// TwinCAT 3 PLC project SortingMashine
// ProgramVersion: 3.1.4023.0
// libraries:
//   Tc2_Standard, * (Beckhoff Automation GmbH)
//   Tc2_System, * (Beckhoff Automation GmbH)
//   Tc3_Module, * (Beckhoff Automation GmbH)
// project tree:
//   DUTs/ Material_Type.TcDUT, Positions.TcDUT
//   / GlobalTextList.TcGTLO, PlcTask.TcTTO, Visualization Manager.TcVMO (not stored)
//   POUs/ FB_Axes.TcPOU, FB_Box.TcPOU, FB_Gate.TcPOU, MAIN.TcPOU, Mashine.TcPOU
//   VISUs/ Visualization.TcVIS
// real-time tasks:
//   TASK PlcTask: cycle T#10ms, priority 20, ADS port 350

CONFIGURATION SortingMashine
    RESOURCE PLC ON TwinCAT3
        TASK PlcTask(INTERVAL := T#10ms, PRIORITY := 20);
        PROGRAM MAIN WITH PlcTask : MAIN;
    END_RESOURCE
END_CONFIGURATION

// ---- DUTs/Material_Type.TcDUT
{attribute 'qualified_only'}
{attribute 'strict'}
TYPE Material_Type :
(
	Plastic := 0,
	Metal :=1
);
END_TYPE

// ---- DUTs/Positions.TcDUT
{attribute 'qualified_only'}
{attribute 'strict'}
TYPE Positions :
(
	First := 180,
	Second:=148,
	Third:=116,
	Forth:=84
);
END_TYPE

// ---- POUs/MAIN.TcPOU
PROGRAM MAIN
VAR
	Mashine1Boxes:ARRAY[1..4] OF FB_Box;
	Mashine2Boxes:ARRAY[1..4] OF FB_Box;
	MyMashine1:Mashine;
	MyMashine2:Mashine;
END_VAR

Mashine1Boxes[1](material:=Material_Type.Plastic);
Mashine1Boxes[2](material:=Material_Type.Metal);
Mashine1Boxes[3](material:=Material_Type.Plastic);
Mashine1Boxes[4](material:=Material_Type.Metal);
Mashine2Boxes[1](material:=Material_Type.Metal);
Mashine2Boxes[2](material:=Material_Type.Plastic);
Mashine2Boxes[3](material:=Material_Type.Metal);
Mashine2Boxes[4](material:=Material_Type.Plastic);

MyMashine1(Box:=Mashine1Boxes);
MyMashine2(Box:=Mashine2Boxes);

END_PROGRAM

// ---- POUs/FB_Box.TcPOU
FUNCTION_BLOCK FB_Box
VAR_INPUT
		material : Material_Type;
		PositionHOZ : INT;
		PositionVTK : INT;
END_VAR
VAR_OUTPUT
END_VAR
VAR
	IsMetal:BOOL;
END_VAR

M_Identify_Material();

METHOD M_Identify_Material : BOOL
VAR_INPUT
END_VAR
IF material=Material_Type.Metal THEN
	IsMetal:=TRUE;
ELSE
	IsMetal:=FALSE;
END_IF
END_METHOD

END_FUNCTION_BLOCK

// ---- POUs/Mashine.TcPOU
FUNCTION_BLOCK Mashine 
VAR_INPUT
	Box:REFERENCE TO ARRAY[1..4] OF FB_Box;
END_VAR
VAR_OUTPUT
END_VAR
VAR
	Current:INT:=1;
	MyGate:FB_Gate;
	FirstAxes:FB_Axes;
	SecondAxes:FB_Axes;
	Step_Stat:INT;
	Step_Stat2:INT;
	Step_Stat3:INT;
END_VAR

CASE Step_Stat OF
	
	0:
		IF OpenGate() THEN
			Step_Stat:=Step_Stat+1;
		END_IF
	1:
		IF MoveOut(Box[Current]) THEN
			Step_Stat:=Step_Stat+1;
		END_IF
	2:
		IF CloseGate()  THEN
			Step_Stat:=Step_Stat+1;
		END_IF
	3:
		IF MoveToFirstPosition(Box[Current])  THEN
			Step_Stat:=Step_Stat+1;
		END_IF
	4:
		IF NOT Box[Current].IsMetal THEN
			IF ExtendFirstAxes(Box[Current]) THEN
				IF Current <4 THEN
					Current:=Current+1;
					Step_Stat:=0;
				ELSE
					Step_Stat:=7;
				END_IF
			END_IF
		ELSE
			Step_Stat:=Step_Stat+1;
		END_IF
	5:
		IF MoveToSecondPosition(Box[Current]) THEN
			Step_Stat:=Step_Stat+1;
		END_IF
	6:
		IF Box[Current].IsMetal THEN
			IF ExtendSecondAxes(Box[Current]) THEN
				IF Current <4 THEN
					Current:=Current+1;
					Step_Stat:=0;
				ELSE
					Step_Stat:=7;
				END_IF
			END_IF
		END_IF
	7://End
		
END_CASE

METHOD CloseGate : BOOL
VAR_INPUT
END_VAR
IF MyGate.GateStat = TRUE THEN
MyGate.GateTimer(IN:=TRUE,PT:=T#1S);	
	IF MyGate.GatePosition > 0 THEN
		MyGate.GatePosition:=MyGate.GatePosition-1;
	END_IF
	IF MyGate.GateTimer.Q THEN		
		MyGate.GateTimer(IN:=FALSE);	
		MyGate.GateStat:=FALSE;
		CloseGate:=TRUE;	
	END_IF	
END_IF
END_METHOD

METHOD ExtendFirstAxes : BOOL
VAR_INPUT
	Box:reference to FB_Box;
END_VAR
CASE FirstAxes.Axes_Step OF
	0:
		IF  FirstAxes.AxesPosition > -55 THEN
			FirstAxes.AxesPosition:= FirstAxes.AxesPosition-1;
			Box.PositionVTK:=Box.PositionVTK-4;
			IF  FirstAxes.AxesPosition <= -55 AND Box.PositionVTK <= -200 THEN
				FirstAxes.Axes_Step:=FirstAxes.Axes_Step+1;
			END_IF
		END_IF		
	1: 
		IF  FirstAxes.AxesPosition < 0 THEN	
			FirstAxes.AxesPosition:= FirstAxes.AxesPosition+1;
			IF  FirstAxes.AxesPosition = 0 THEN
				ExtendFirstAxes:=TRUE;
				FirstAxes.Axes_Step:=0;
			END_IF		
		END_IF
END_CASE	







//IF FirstAxes.Extended = FALSE THEN
//	IF  FirstAxes.AxesPosition > -55 THEN
//		 FirstAxes.AxesPosition:= FirstAxes.AxesPosition-1;
//	END_IF	
	
//	IF  FirstAxes.AxesPosition = -55 THEN
		
//			FirstAxes.Extended:=TRUE;
//		 	FirstAxes.AxesTimer(IN:=TRUE,PT:=T#500MS);
//		IF FirstAxes.AxesTimer.Q AND  FirstAxes.Extended:=TRUE THEN
			
//			IF  FirstAxes.AxesPosition < 0 THEN
//				 FirstAxes.AxesPosition:= FirstAxes.AxesPosition+1;
//			END_IF
	
//			IF  FirstAxes.AxesPosition = 0 THEN
//				FirstAxes.AxesTimer(IN:=FALSE);
//				FirstAxes.Extended:=FALSE;
//			END_IF
			
//		END_IF
		
//	END_IF
	
//END_IF
END_METHOD

METHOD ExtendSecondAxes : BOOL
VAR_INPUT
	Box:REFERENCE TO FB_Box;
END_VAR
CASE SecondAxes.Axes_Step OF
	0: 
		IF  SecondAxes.AxesPosition > -55 THEN
			SecondAxes.AxesPosition:= SecondAxes.AxesPosition-1;
			Box.PositionVTK:=Box.PositionVTK-4;
			IF  SecondAxes.AxesPosition <= -55 AND Box.PositionVTK <= -200 THEN
				SecondAxes.Axes_Step:=SecondAxes.Axes_Step+1;
			END_IF
		END_IF		
	1: 
		IF  SecondAxes.AxesPosition < 0 THEN	
			SecondAxes.AxesPosition:= SecondAxes.AxesPosition+1;
			IF  SecondAxes.AxesPosition = 0 THEN
				ExtendSecondAxes:=TRUE;
				SecondAxes.Axes_Step:=0;
			END_IF		
		END_IF
END_CASE
END_METHOD

METHOD MoveOut : BOOL
VAR_INPUT
	Box: reference to FB_Box;
END_VAR
IF Box.PositionHOZ < 50 THEN
Box.PositionHOZ:=Box.PositionHOZ+1;	
	IF Box.PositionHOZ = 50 THEN
		MoveOut:=TRUE;		
	END_IF
ELSIF Box.PositionHOZ = 50 THEN
	MoveOut:=TRUE;
END_IF
END_METHOD

METHOD MoveToFirstPosition : BOOL
VAR_INPUT
	Box:reference to FB_Box;
END_VAR
IF Box.PositionHOZ < 483 THEN
Box.PositionHOZ:=Box.PositionHOZ+1;	
	IF Box.PositionHOZ=483 THEN
		MoveToFirstPosition:=TRUE;			
	END_IF	
END_IF
END_METHOD

METHOD MoveToSecondPosition : BOOL
VAR_INPUT
	Box:reference to FB_Box;
END_VAR
IF Box.PositionHOZ < 685 THEN
Box.PositionHOZ:=Box.PositionHOZ+1;	
	IF Box.PositionHOZ=685 THEN
		MoveToSecondPosition:=TRUE;			
	END_IF	
END_IF
END_METHOD

METHOD OpenGate : BOOL
VAR_INPUT
END_VAR
VAR
	i:INT;
	
END_VAR
IF MyGate.GateStat = FALSE THEN
	MyGate.GateTimer(IN:=TRUE,PT:=T#1S);	
	IF MyGate.GatePosition < 50 THEN
		MyGate.GatePosition:=MyGate.GatePosition+1;
	END_IF
	IF MyGate.GateTimer.Q AND MyGate.GatePosition >=50 THEN		
			MyGate.GateTimer(IN:=FALSE);	
			MyGate.GateStat:=TRUE;
			OpenGate:=TRUE;	
	END_IF	
END_IF
END_METHOD

END_FUNCTION_BLOCK

// ---- POUs/FB_Gate.TcPOU
FUNCTION_BLOCK FB_Gate
VAR_INPUT
	GateStat:BOOL;
	GatePosition:INT;
	GateTimer:TON;
END_VAR

END_FUNCTION_BLOCK

// ---- POUs/FB_Axes.TcPOU
FUNCTION_BLOCK FB_Axes
VAR_INPUT
	AxesPosition:INT;
	Extended:BOOL;
	Axes_Step:Int:=0;
END_VAR
VAR
END_VAR

END_FUNCTION_BLOCK

// ---- VISUs/Visualization.TcVIS
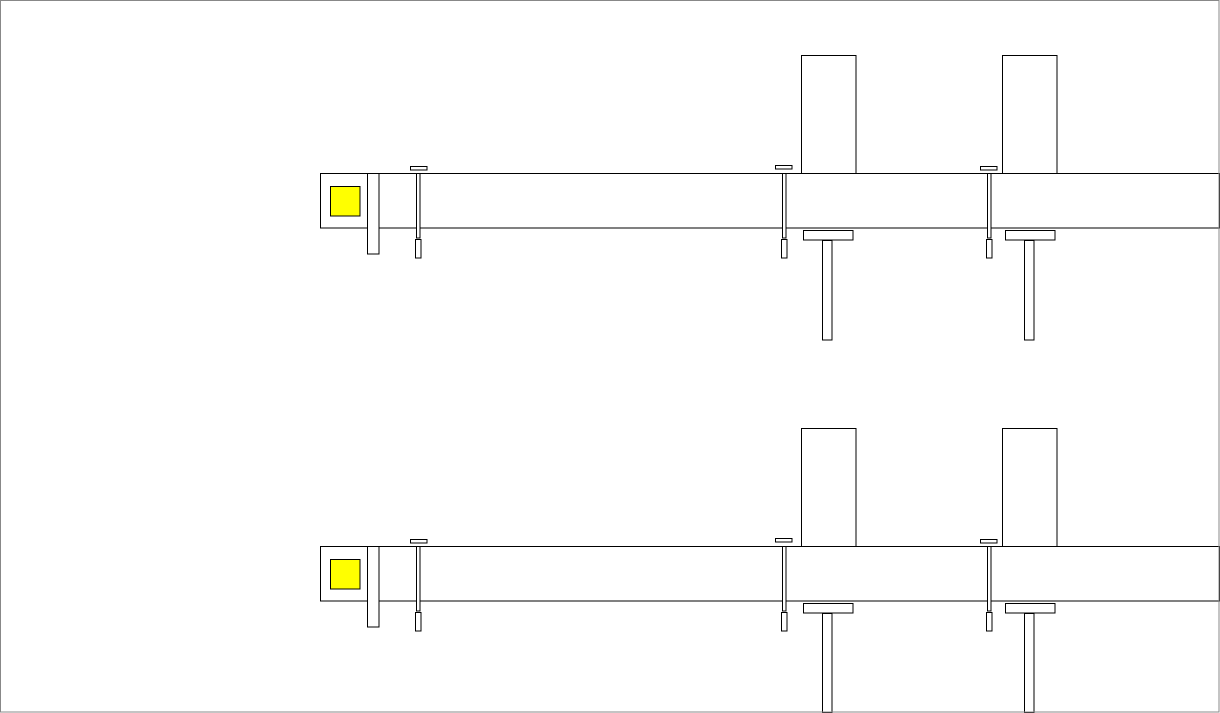
VISUALIZATION Visualization  // 1220x713
    Rectangle (801,55 55x120)
    Rectangle (1002,55 55x120)
    Rectangle (320,173 900x55)
    Rectangle (330,186 30x30), colour toggle: MAIN.Mashine1Boxes[4].IsMetal
        p3560616238: MAIN.Mashine1Boxes[4].PositionHOZ
        p2738717112: MAIN.Mashine1Boxes[4].PositionVTK
    Rectangle (330,186 30x30), colour toggle: MAIN.Mashine1Boxes[3].IsMetal
        p3560616238: MAIN.Mashine1Boxes[3].PositionHOZ
        p2738717112: MAIN.Mashine1Boxes[3].PositionVTK
    Group (803,230 50x110)
        p2738717112: MAIN.MyMashine1.FirstAxes.AxesPosition
        Rectangle (0,0 50x10)
        Rectangle (19,10 10x100)
    Group (1005,230 50x110)
        p2738717112: MAIN.MyMashine1.SecondAxes.AxesPosition
        Rectangle (0,0 50x10)
        Rectangle (19,10 10x100)
    Rectangle (330,186 30x30), colour toggle: MAIN.Mashine1Boxes[2].IsMetal
        p3560616238: MAIN.Mashine1Boxes[2].PositionHOZ
        p2738717112: MAIN.Mashine1Boxes[2].PositionVTK
    Rectangle (416,173 4x65)
    Rectangle (782,173 4x65)
    Rectangle (987,173 4x65)
    Rectangle (367,173 12x81)
        p2738717112: MAIN.MyMashine1.MyGate.GatePosition
    Rectangle (410,166 17x4)
    Rectangle (775,165 17x4)
    Rectangle (980,166 17x4)
    Rectangle (415,239 6x19)
    Rectangle (781,239 6x19)
    Rectangle (986,239 6x19)
    Rectangle (330,186 30x30), colour toggle: MAIN.Mashine1Boxes[1].IsMetal
        p3560616238: MAIN.Mashine1Boxes[1].PositionHOZ
        p2738717112: MAIN.Mashine1Boxes[1].PositionVTK
    Rectangle (801,428 55x120)
    Rectangle (1002,428 55x120)
    Rectangle (320,546 900x55)
    Rectangle (330,559 30x30), colour toggle: MAIN.Mashine2Boxes[4].IsMetal
        p3560616238: MAIN.Mashine2Boxes[4].PositionHOZ
        p2738717112: MAIN.Mashine2Boxes[4].PositionVTK
    Rectangle (330,559 30x30), colour toggle: MAIN.Mashine2Boxes[3].IsMetal
        p3560616238: MAIN.Mashine2Boxes[3].PositionHOZ
        p2738717112: MAIN.Mashine2Boxes[3].PositionVTK
    Group (803,603 50x110)
        p2738717112: MAIN.MyMashine2.FirstAxes.AxesPosition
        Rectangle (0,0 50x10)
        Rectangle (19,10 10x100)
    Group (1005,603 50x110)
        p2738717112: MAIN.MyMashine2.SecondAxes.AxesPosition
        Rectangle (0,0 50x10)
        Rectangle (19,10 10x100)
    Rectangle (330,559 30x30), colour toggle: MAIN.Mashine2Boxes[2].IsMetal
        p3560616238: MAIN.Mashine2Boxes[2].PositionHOZ
        p2738717112: MAIN.Mashine2Boxes[2].PositionVTK
    Rectangle (416,546 4x65)
    Rectangle (782,546 4x65)
    Rectangle (987,546 4x65)
    Rectangle (367,546 12x81)
        p2738717112: MAIN.MyMashine2.MyGate.GatePosition
    Rectangle (410,539 17x4)
    Rectangle (775,538 17x4)
    Rectangle (980,539 17x4)
    Rectangle (415,612 6x19)
    Rectangle (781,612 6x19)
    Rectangle (986,612 6x19)
    Rectangle (330,559 30x30), colour toggle: MAIN.Mashine2Boxes[1].IsMetal
        p3560616238: MAIN.Mashine2Boxes[1].PositionHOZ
        p2738717112: MAIN.Mashine2Boxes[1].PositionVTK
END_VISUALIZATION
